(* PLC project KinIn_v3.project, CODESYS CODESYS V3.5 SP19 *)
(* stored: creationDateTime 2025-01-20T16:26:49.2807479, modificationDateTime 2025-01-20T16:17:39.6822999 *)

FUNCTION_BLOCK TransSE3_ToRotAndPos
  VAR_INPUT
    T : ARRAY[1..4, 1..4] OF REAL;  (* transform *)
  END_VAR
  VAR_OUTPUT
    RotMat : ARRAY[1..3, 1..3] OF REAL;  (* rotation matrix *)
    p : ARRAY[1..3] OF REAL;  (* position array *)
  END_VAR
  VAR
    i : DINT;
    j : DINT;
  END_VAR

            i:=1;j:=1;
FOR i:=1 TO 3 DO
	FOR j:=1 TO 3 DO
		RotMat[i,j]:=T[i,j];//equals to RotMatrix
	END_FOR
END_FOR

p[1]:=T[1,4];
p[2]:=T[2,4];
p[3]:=T[3,4];
          
END_FUNCTION_BLOCK
